(* IEC 61131-3 sources: AXOpen/src/components.robotics/ctrl/src/AxoRobotics, 4 files *)

(* ---- CalculateDistance.st ---- *)
USING System.Math;

NAMESPACE AXOpen.Components.Robotics
    FUNCTION CalculateDistance : REAL
        VAR_INPUT
            inDistType : AXOpen.Components.Abstractions.Robotics.eAxoRoboticsDistance;
            inP1 : AXOpen.Components.Abstractions.Robotics.AxoRoboticsCoordinates;
            inP2 : AXOpen.Components.Abstractions.Robotics.AxoRoboticsCoordinates;
        END_VAR
        VAR
            x2 : REAL;
            y2 : REAL;
            z2 : REAL;
        END_VAR
        x2 := (inP1.X-inP2.X);
        x2 := x2 * x2;
        y2 := (inP1.Y-inP2.Y);
        y2 := y2 * y2;
        z2 := (inP1.Z-inP2.Z);
        z2 := z2 * z2;
        CASE inDistType OF
            AXOpen.Components.Abstractions.Robotics.eAxoRoboticsDistance#X:
                CalculateDistance := SQRT(x2);
            AXOpen.Components.Abstractions.Robotics.eAxoRoboticsDistance#Y:
                CalculateDistance := SQRT(y2);
            AXOpen.Components.Abstractions.Robotics.eAxoRoboticsDistance#Z:
                CalculateDistance := SQRT(z2);
            AXOpen.Components.Abstractions.Robotics.eAxoRoboticsDistance#XY:
                CalculateDistance := SQRT(x2+y2);
            AXOpen.Components.Abstractions.Robotics.eAxoRoboticsDistance#XZ:
                CalculateDistance := SQRT(x2+z2);
            AXOpen.Components.Abstractions.Robotics.eAxoRoboticsDistance#YZ:
                CalculateDistance := SQRT(y2+z2);
            AXOpen.Components.Abstractions.Robotics.eAxoRoboticsDistance#XYZ:
                CalculateDistance := SQRT(x2+y2+z2);
        END_CASE;
    END_FUNCTION
END_NAMESPACE

(* ---- CoordinatesAreNearlyEqual.st ---- *)
USING System.Math;

NAMESPACE AXOpen.Components.Robotics
    FUNCTION CoordinatesAreNearlyEqual : BOOL
        VAR_IN_OUT
            Coordinates1 : AXOpen.Components.Abstractions.Robotics.AxoRoboticsCoordinates;
            Coordinates2 : AXOpen.Components.Abstractions.Robotics.AxoRoboticsCoordinates;
        END_VAR
        VAR_INPUT
            EpsilonX : REAL;
            EpsilonY : REAL;
            EpsilonZ : REAL;
            EpsilonRx : REAL;
            EpsilonRy : REAL;
            EpsilonRz : REAL;
        END_VAR

        CoordinatesAreNearlyEqual :=	IsNearlyEqual(Coordinates1.X,Coordinates2.X,EpsilonX)  AND
                                        IsNearlyEqual(Coordinates1.Y,Coordinates2.Y,EpsilonY)  AND
                                        IsNearlyEqual(Coordinates1.Z,Coordinates2.Z,EpsilonZ)  AND
                                        IsNearlyEqual(Coordinates1.Rx,Coordinates2.Rx,EpsilonRx)  AND
                                        IsNearlyEqual(Coordinates1.Ry,Coordinates2.Ry,EpsilonRy)  AND
                                        IsNearlyEqual(Coordinates1.Rz,Coordinates2.Rz,EpsilonRz);
    END_FUNCTION
END_NAMESPACE

(* ---- IsNearlyEqual.st ---- *)
USING System.Math;

NAMESPACE AXOpen.Components.Robotics
    FUNCTION IsNearlyEqual : BOOL
        VAR_INPUT
            Coordinate1 : REAL;
            Coordinate2 : REAL;
            Epsilon : REAL;
        END_VAR
        VAR
            AbsCoordinate1 : REAL;
            AbsCoordinate2 : REAL;
            Diff : REAL;
            Denominator : LREAL;
        END_VAR
        IsNearlyEqual := FALSE;
        AbsCoordinate1 := ABS(Coordinate1);
        AbsCoordinate2 := ABS (Coordinate2);
        Diff := ABS(Coordinate1-Coordinate2) ;
        Denominator := AbsCoordinate1;
        Denominator := Denominator + AbsCoordinate2;

        IF Epsilon < 0 THEN
            RETURN;
        END_IF;

        IF Coordinate1 = Coordinate2 THEN
            IsNearlyEqual := TRUE;
        ELSIF (Coordinate1 = 0 OR Coordinate2 = 0) AND Diff <= Epsilon THEN
            IsNearlyEqual := Diff <= Epsilon;
        ELSE
            IsNearlyEqual := Diff / Denominator <= Epsilon;
        END_IF;

    END_FUNCTION
END_NAMESPACE

(* ---- AxoRobot_Status.st ---- *)
USING AXOpen.Core;
NAMESPACE AXOpen.Components.Robotics
    {#ix-attr:[Container(Layout.Stack)]}
    {S7.extern=ReadWrite}
    CLASS AxoRobot_Status EXTENDS AXOpen.Components.Abstractions.AxoComponent_Status
        VAR PUBLIC
            {#ix-set:AttributeName = "<#Current movement parameters#>"}
            {#ix-attr:[ReadOnly()]}
            CurrentMovementParameters    :   AXOpen.Components.Abstractions.Robotics.AxoRoboticsMovementsParams;
        END_VAR
    END_CLASS
END_NAMESPACE
